# B&R Automation Studio project MatveevK.A-KRBO-02-17-Lab3
Automation Studio 4.5.2.102

## Logical view

Binary libraries used (declarations not repeated): Runtime, Operator, AsIecCon, astime, sys_lib, asstring, Acp10man, Acp10par, NcGlobal, Acp10sdc, Acp10_MC, brsystem, AsBrStr, Acp10sim, AsIOTime

### Library Logical/MotrContr (ANSIC)

#### Types.typ
```iecst
TYPE
	axis_states :
		(
		B,
		B_dir,
		A,
		A_dir,
		unknown
		);
END_TYPE
```

#### MotrContr.fun
```iecst
{REDUND_ERROR} {REDUND_UNREPLICABLE} FUNCTION_BLOCK FB_Integrator (*TODO: Add your comment here*) (*$GROUP=User,$CAT=User,$GROUPICON=User.png,$CATICON=User.png*)
	VAR_INPUT
		in : {REDUND_UNREPLICABLE} REAL;
	END_VAR
	VAR_OUTPUT
		out : {REDUND_UNREPLICABLE} REAL;
	END_VAR
	VAR
		dt : {REDUND_UNREPLICABLE} REAL;
	END_VAR
END_FUNCTION_BLOCK

{REDUND_ERROR} {REDUND_UNREPLICABLE} FUNCTION_BLOCK FB_Motor (*TODO: Add your comment here*) (*$GROUP=User,$CAT=User,$GROUPICON=User.png,$CATICON=User.png*)
	VAR_INPUT
		u : {REDUND_UNREPLICABLE} REAL;
	END_VAR
	VAR_OUTPUT
		w : {REDUND_UNREPLICABLE} REAL;
		phi : {REDUND_UNREPLICABLE} REAL;
	END_VAR
	VAR
		integrator : {REDUND_UNREPLICABLE} FB_Integrator;
		Tm : {REDUND_UNREPLICABLE} REAL;
		ke : {REDUND_UNREPLICABLE} REAL;
		dt : {REDUND_UNREPLICABLE} REAL;
	END_VAR
END_FUNCTION_BLOCK

{REDUND_ERROR} FUNCTION_BLOCK FB_Regulator (*TODO: Add your comment here*) (*$GROUP=User,$CAT=User,$GROUPICON=User.png,$CATICON=User.png*)
	VAR_INPUT
		e : {REDUND_UNREPLICABLE} REAL;
	END_VAR
	VAR_OUTPUT
		u : {REDUND_UNREPLICABLE} REAL;
	END_VAR
	VAR
		k_p : {REDUND_UNREPLICABLE} REAL;
		k_i : {REDUND_UNREPLICABLE} REAL;
		integrator : {REDUND_UNREPLICABLE} FB_Integrator;
		iyOld : {REDUND_UNREPLICABLE} REAL;
		max_abs_value : {REDUND_UNREPLICABLE} REAL;
		abs_in_2 : REAL;
		abs_in_1 : REAL;
		abs_out_1 : REAL;
		e_kp : REAL;
		dt : {REDUND_UNREPLICABLE} REAL;
	END_VAR
END_FUNCTION_BLOCK

{REDUND_ERROR} FUNCTION_BLOCK FB_Axis (*TODO: Add your comment here*) (*$GROUP=User,$CAT=User,$GROUPICON=User.png,$CATICON=User.png*)
	VAR_INPUT
		reset_error : BOOL;
		endswitch_a_reached : BOOL;
		endswitch_b_reached : BOOL;
		u : REAL;
		button_a : BOOL;
		button_b : BOOL;
		direction : BOOL;
		state : INT;
	END_VAR
	VAR_OUTPUT
		reset_counter : BOOL;
		pwm_value : INT;
		counter : INT;
		speed : REAL;
	END_VAR
	VAR
		last_counter : INT;
	END_VAR
END_FUNCTION_BLOCK
```

#### FB_Axis.c
```c
#include <bur/plctypes.h>
#ifdef __cplusplus
	extern "C"
	{
#endif
	#include "MotrContr.h"
#ifdef __cplusplus
	};
#endif
/* TODO: Add your comment here */
void FB_Axis(struct FB_Axis* inst)
{

	/*
	switch(inst->state)
	{
		case unknown:
			if (inst->endswitch_a_reached || inst->button_a)
				inst->state = A;

			if (inst->endswitch_b_reached || inst->button_b)
				inst->state = B;

			if (inst->direction)								//
				inst->state = A_dir;

			if (!inst->direction)								//
				inst->state = B_dir;

			break;

		case B:
			inst->pwm_value = 0;
			inst->reset_error = 1;

			if (!inst->button_b && !inst->endswitch_b_reached)
				inst->state = B_dir;

			if (inst->direction)								//
				inst->state = A_dir;
			break;

		case A:
			inst->pwm_value = 0;
			inst->reset_error = 1;

			if (!inst->button_a && !inst->endswitch_a_reached)
				inst->state = A_dir;

			if (!inst->direction)								//
				inst->state = B_dir;
			break;

		case A_dir:
			inst->pwm_value = inst->u / 24.0 * 32767;			//шим соответственно напряжению с регулятора
			inst->reset_error = 0;
			inst->speed = inst->u / 24.0 * 6500.0;

			if (inst->endswitch_a_reached || inst->button_a)
				inst->state = A;

			if (!inst->direction)								//
				inst->state = B_dir;

			break;

		case B_dir:
			inst->pwm_value = -inst->u / 24.0 * 32767;			//шим соответственно напряжению с регулятора
			inst->reset_error = 0;
			inst->speed = -inst->u / 24.0 * 6500.0;

			if (inst->endswitch_b_reached || inst->button_b)
				inst->state = B;

			if (inst->direction)								//
				inst->state = A_dir;

			break;
	}
	*/

	/*if (inst->endswitch_a_reached || inst->endswitch_b_reached)
	{
		inst->reset_error=1;
	}
	else
	{*/
		inst->pwm_value=inst->u / 24.0 * 32767;//шим соответственно напряжению с регулятора
		//inst->reset_error=0;
	///}
	inst->speed = inst->u / 24.0 * 6500.0;
}
```

#### FB_Integrator.c
```c
#include <bur/plctypes.h>
#ifdef __cplusplus
	extern "C"
	{
#endif
	#include "MotrContr.h"
#ifdef __cplusplus
	};
#endif
/* TODO: Add your comment here */
void FB_Integrator(struct FB_Integrator* inst)
{
	inst->out += inst->in * inst->dt;
}
```

#### FB_Regulator.c
```c
#include <bur/plctypes.h>
#ifdef __cplusplus
	extern "C"
	{
#endif
#include "MotrContr.h"
#include "Math.h"				///////////////////////
#ifdef __cplusplus
	};
#endif
/* TODO: Add your comment here */
void FB_Regulator(struct FB_Regulator* inst)
{
	/*
	inst->integrator.in=inst->e * inst->k_i * inst->dt + inst->iyOld;

	FB_Integrator(&(inst->integrator));

	inst->e_kp=inst->e*inst->k_p;

	inst->e_kp=(inst->e_kp > inst->max_abs_value || inst->e_kp < - inst->max_abs_value)?((inst->e_kp>0)?inst->max_abs_value:-inst->max_abs_value):inst->e_kp;

	inst->e_kp+=inst->integrator.out;

	inst->u=(inst->e_kp > inst->max_abs_value || inst->e_kp < - inst->max_abs_value)?((inst->e_kp>0)?inst->max_abs_value:-inst->max_abs_value):inst->e_kp;

	inst->iyOld=inst->u-inst->e_kp;
	*/

	inst->integrator.in = inst->k_i * inst->e + inst->iyOld / inst->dt;
	FB_Integrator(&inst->integrator);
	if(fabs(inst->k_p * inst->e) < inst->max_abs_value)
	{
		inst->e_kp = inst->e * inst->k_p + inst->integrator.out;
	}
	else
	{
		//BOOL a = 1;
		inst->e_kp = inst->max_abs_value * copysign(1.0, inst->k_p * inst->e) + inst->integrator.out;
	}
	if(fabs(inst->e_kp) < inst->max_abs_value)
	{
		inst->u = inst->e_kp;
	}
	else
	{
		inst->u = inst->max_abs_value * copysign(1.0, inst->e_kp);
	}
	inst->iyOld = inst->u - inst->e_kp;
}
```

### Program Logical/SDCAxisCtrlX

#### Cyclic.c
```c
#include <bur/plctypes.h>

#ifdef _DEFAULT_INCLUDES
	#include <AsDefault.h>
#endif

void _CYCLIC ProgramCyclic(void)
{
	gAxis_X_EncIf.iLifeCnt++;
	gAxis_X_DiDoIf.iLifeCntDriveEnable++;
	gAxis_X_DiDoIf.iLifeCntDriveReady++;
	gAxis_X_DiDoIf.iLifeCntNegHwEnd++;
	gAxis_X_DiDoIf.iLifeCntPosHwEnd++;
	gAxis_X_DiDoIf.iLifeCntReference++;
	gAxis_X_DrvIf.iLifeCnt++;

	gAxis_X_EncIf.iActTime = (INT)AsIOTimeCyclicStart();
	gAxis_X_EncIf.iActPos = axis_X.counter;

	gAxis_X_DiDoIf.iPosHwEnd = axis_X.endswitch_a_reached;
	gAxis_X_DiDoIf.iNegHwEnd = axis_X.endswitch_b_reached;

	//coil_pwm_value = coil_powered?32767:0;
	if(coil_powered)
		coil_pwm_value = 32767;
	else
		coil_pwm_value = 0;

	//fb_controller.e = 100 * 6500.0 / 32767 - axis_X.speed; //6500.0 максимльня скорость в метках в секунду
	fb_controller.e = gAxis_X_DrvIf.oSetPos * 6500 / 32767 - axis_X.speed; //6500.0 максимльня скорость в метках в секунду
	FB_Regulator(&fb_controller); // передать значение в регулятор
	axis_X.u = fb_controller.u;

	//axis_X.u = 18;

	FB_Axis(&axis_X);
}
```

#### Init.c
```c
#include <bur/plctypes.h>

#ifdef _DEFAULT_INCLUDES
	#include <AsDefault.h>
#endif

void _INIT ProgramInit(void)
{
	//Устанавливаем типы SDC модулей
	gAxis_X_HW.EncIf1_Typ = ncSDC_ENC16;
	gAxis_X_HW.DiDoIf_Typ = ncSDC_DIDO;
	gAxis_X_HW.DrvIf_Typ = ncSDC_DRVSERVO16;
	//Устанавливаем имена переменных
	strcpy(gAxis_X_HW.EncIf1_Name, "gAxis_X_EncIf");
	strcpy(gAxis_X_HW.DrvIf_Name, "gAxis_X_DrvIf");
	strcpy(gAxis_X_HW.DiDoIf_Name, "gAxis_X_DiDoIf");
	//Устанавливаем входы готовности и нормальной работы
	gAxis_X_EncIf.iEncOK = 1;
	gAxis_X_DrvIf.iDrvOK = 1;
	gAxis_X_DrvIf.iStatusEnable = 1;
	gAxis_X_DiDoIf.iDriveReady = 1;

	fb_controller.k_p=0.002;
	fb_controller.k_i=0.16;

	fb_controller.dt=0.002;
	fb_controller.integrator.dt=0.002;

	fb_controller.max_abs_value=24;

	pwm_period = 200;

	enable=1;
}
```
